PROGRAM SafetyHandling
VAR
	restart_safety 	: TP;
	//safety_state 	: RS;
	start_delay 	: TON;
	ErrAck_Pulse	: TP;
	SafetyLog		: FB_EventLog;
END_VAR
VAR_OUTPUT
	Error			: BOOL;
END_VAR

// Safety can be stopped by pressing STOP and RESET on main panel
GVL_Safety.Run := GVL_Main.phase_available AND NOT (GVL_Main.stop_switch AND GVL_Main.reset_switch);
// power on delay for Safety RESTART after RUN=1
restart_safety(IN := GVL_Main.phase_available, PT := T#1S);
// RESTART Safety after pushing reset or power on delay
GVL_Safety.Restart := Main.reset OR restart_safety.Q;

// wait n seconds after Start ...
start_delay(IN := GVL_Main.phase_available, PT := T#15S);
// ... and send ErrAck for n milliseconds
ErrAck_Pulse(IN := GVL_Main.phase_available AND start_delay.Q, PT := T#200MS);

// Error Acknowledgment: Turn key_switch OFF and press STOP 
GVL_Safety.ErrAck := (NOT GVL_Main.key_switch_remote AND GVL_Main.stop_switch)
					OR (NOT GVL_pendant_control.key_switch AND GVL_pendant_control.reset_switch)
					OR ErrAck_Pulse.Q;
Error := GVL_Safety.Error;

SafetyLog(Trigger := Error,
				Level := ADSLOG_MSGTYPE_ERROR,
				OnMessage := 'Safety Error! Emergency stop enganged!',
				OffMessage := 'Safety is OK.',
				OffLevel := ADSLOG_MSGTYPE_HINT);

END_PROGRAM

(* stored: Version 1.1.0.1, ProductVersion 3.1.4024.9
   POU SafetyHandling: Id {6d4a788c-2168-4769-93de-c67314036861}, SpecialFunc None *)
